SUBAPPLICATION Uebung_016b_AX (* Background Colour umschalten -- 3-fach mit SubApp *)
  (* Standard: 61499-2; Description: Copyright (c) 2026 Meisterschulen am Ostbahnhof This program and the accompanying materials are made available under the terms of the Eclipse Public License 2.0 which is available at https://www.eclipse.org/legal/epl-2.0/ SPDX-License-Identifier: EPL-2.0 *)
  (* Version 1.0, 2026-09-10, Franz Höpfinger, Meisterschulen am Ostbahnhof, initial API and implementation and/or initial documentation *)
  PACKAGE Uebungen;
  IMPORT isobus::UT::io::Softkey::SoftKeyActivationCode::SK_RELEASED;
  IMPORT Uebungen::const::UT::DefaultPool::SoftKey_F1;
  IMPORT Uebungen::const::UT::DefaultPool::SoftKey_F2;
  IMPORT Uebungen::const::UT::DefaultPool::SoftKey_F3;
  IMPORT Uebungen::const::UT::DefaultPool::SoftKey_F7;
  IMPORT isobus::UT::Q::const::colours::COLOR_GREEN;
  IMPORT isobus::UT::Q::const::colours::COLOR_RED;
  IMPORT isobus::UT::Q::const::colours::COLOR_WHITE;
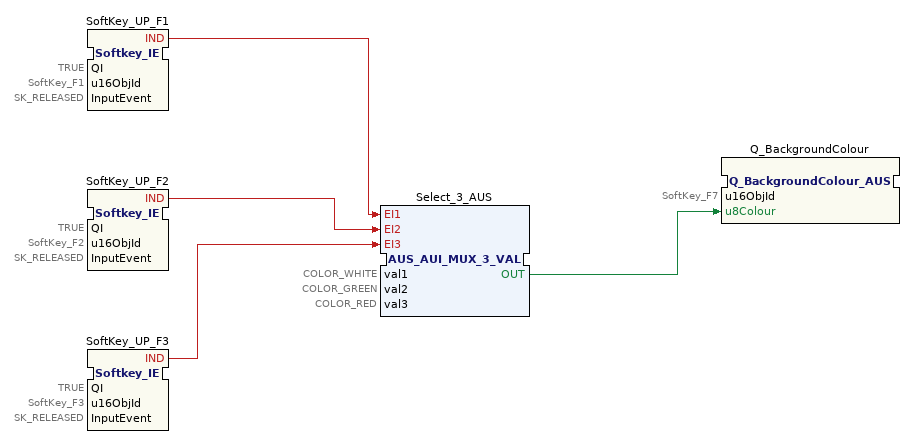
  FBS
    SoftKey_UP_F1 : isobus::UT::io::Softkey::Softkey_IE(QI := TRUE, u16ObjId := SoftKey_F1, InputEvent := SK_RELEASED);
    SoftKey_UP_F2 : isobus::UT::io::Softkey::Softkey_IE(QI := TRUE, u16ObjId := SoftKey_F2, InputEvent := SK_RELEASED);
    SoftKey_UP_F3 : isobus::UT::io::Softkey::Softkey_IE(QI := TRUE, u16ObjId := SoftKey_F3, InputEvent := SK_RELEASED);
    Q_BackgroundColour : isobus::UT::Q::Q_BackgroundColour_AUS(u16ObjId := SoftKey_F7);
  END_FBS
  SUBAPPS
    Select_3_AUS : MyLib::sys::AUS_AUI_MUX_3_VAL(val1 := COLOR_WHITE, val2 := COLOR_GREEN, val3 := COLOR_RED);
  END_SUBAPPS
  EVENT_CONNECTIONS
    SoftKey_UP_F1.IND TO Select_3_AUS.EI1;
    SoftKey_UP_F2.IND TO Select_3_AUS.EI2;
    SoftKey_UP_F3.IND TO Select_3_AUS.EI3;
  END_CONNECTIONS
  ADAPTER_CONNECTIONS
    Select_3_AUS.OUT TO Q_BackgroundColour.u8Colour;
  END_CONNECTIONS
END_SUBAPPLICATION
